INTERFACE itfAutoManual

METHOD mAutoOff : BOOL
VAR_INPUT
END_VAR
END_METHOD

METHOD mAutoOn : BOOL
VAR_INPUT
END_VAR
END_METHOD

METHOD mFault : BOOL
VAR_INPUT
END_VAR
END_METHOD

METHOD mManual : BOOL
VAR_INPUT
END_VAR
END_METHOD

METHOD mRunning : BOOL
VAR_INPUT
END_VAR
END_METHOD

END_INTERFACE

(* stored: Version 1.1.0.1, ProductVersion 3.1.4024.12
   Itf itfAutoManual: Id {b2f36530-f0d8-4d3b-b92b-067f34a2e104}
   Method mAutoOff: Id {58f1948f-8b98-4423-90fe-9664fe275be7}
   Method mAutoOn: Id {bcdee737-f7f3-467a-a5a4-09ca5a410a5d}
   Method mFault: Id {c8fa4e52-e766-484d-8066-f26a7938ddb9}
   Method mManual: Id {2ecbe8c4-fa06-4737-b649-ab0748812381}
   Method mRunning: Id {c2953d72-b0ac-47a7-93af-fea729a9a0b3} *)
